{attribute 'GeneratedUsingTerminal: ELM2644-0000-0016'}
{attribute addProperty BoxType "ELM2644-0000-0016"}
{attribute addProperty Id "Outputs_Channel_3AT %Q*Outputs_Channel_78994C084"}
{attribute addProperty CRC "584924210"}
{attribute addProperty Size "4"}
TYPE DO_Group_3_Outputs_22DD3C32 :
STRUCT
	{attribute addProperty Name "Outputs_Channel_3"}
	Outputs_Channel_3 AT %Q* : Outputs_Channel_78994C08;
END_STRUCT
END_TYPE

(* stored: Version 1.2.0.0, ProductVersion 3.1.4024.9
   DUT DO_Group_3_Outputs_22DD3C32: Id {1d8b8071-dab3-456e-9c9d-8cd12ab97b41} *)
